// TIA Portal V18 export
// export: Created 2026-01-09T11:32:04.0903936Z, ExportSetting WithDefaults, DisplayName Totally Integrated Automation Portal, DisplayVersion V18 Update 5, DisplayName TIA Portal Openness, DisplayVersion V18 Update 5, DisplayName TIA Portal Teamcenter Gateway, DisplayVersion V18, DisplayName TIA Portal Version Control Interface, DisplayVersion V18, DisplayName SINAMICS Startdrive Advanced, DisplayVersion V18 SP2 Update 1, DisplayName SINAMICS Startdrive G110M, G120, G120C, G120D, G120P, G115D, DisplayVersion V18 SP2 Update 1, DisplayName SINAMICS Startdrive G130, G150, S120, S150, SINAMICS MV, S210, G220, S200, DisplayVersion V18 SP2 Update 1, DisplayName STEP 7 Professional, DisplayVersion V18 Update 5, DisplayName STEP 7 Safety, DisplayVersion V18, DisplayName WinCC Professional, DisplayVersion V18 Update 5
TagTable "ST_PM"
  ST_PMDBNum : Int  (1 s)
  ST_PMStepNext{1} : Bool  (%DB[ST_PMDBNum].DBX0.5, CPU S71500-2PN_TP700, 1 s)
  ST_PMStepNext{2} : Bool  (%DB[ST_PMDBNum].DBX20.5, CPU S71500-2PN_TP700, 1 s)
  ST_PMStepNext{3} : Bool  (%DB[ST_PMDBNum].DBX40.5, CPU S71500-2PN_TP700, 1 s)
  ST_PMStepNext{4} : Bool  (%DB[ST_PMDBNum].DBX60.5, CPU S71500-2PN_TP700, 1 s)
  ST_PMStepNext{5} : Bool  (%DB[ST_PMDBNum].DBX80.5, CPU S71500-2PN_TP700, 1 s)
  ST_PMStepNext{6} : Bool  (%DB[ST_PMDBNum].DBX100.5, CPU S71500-2PN_TP700, 1 s)
  ST_PMStepNext{7} : Bool  (%DB[ST_PMDBNum].DBX120.5, CPU S71500-2PN_TP700, 1 s)
  ST_PMStepNext{8} : Bool  (%DB[ST_PMDBNum].DBX140.5, CPU S71500-2PN_TP700, 1 s)
  ST_PMStepNext{9} : Bool  (%DB[ST_PMDBNum].DBX160.5, CPU S71500-2PN_TP700, 1 s)
  ST_PMStepNext{10} : Bool  (%DB[ST_PMDBNum].DBX180.5, CPU S71500-2PN_TP700, 1 s)
  ST_PMStepNext{11} : Bool  (%DB[ST_PMDBNum].DBX200.5, CPU S71500-2PN_TP700, 1 s)
  ST_PMStepNext{12} : Bool  (%DB[ST_PMDBNum].DBX220.5, CPU S71500-2PN_TP700, 1 s)
  ST_PMStepNext{13} : Bool  (%DB[ST_PMDBNum].DBX240.5, CPU S71500-2PN_TP700, 1 s)
  ST_PMStepNext{14} : Bool  (%DB[ST_PMDBNum].DBX260.5, CPU S71500-2PN_TP700, 1 s)
  ST_PMStepNext{15} : Bool  (%DB[ST_PMDBNum].DBX280.5, CPU S71500-2PN_TP700, 1 s)
  ST_PMStepNext{16} : Bool  (%DB[ST_PMDBNum].DBX300.5, CPU S71500-2PN_TP700, 1 s)
  ST_PMOperatorPrompt[0] : UInt  (%DB[ST_PMDBNum].DBW10, CPU S71500-2PN_TP700, 500 ms)
  ST_PMOperatorPrompt[1] : UInt  (%DB[ST_PMDBNum].DBW10, CPU S71500-2PN_TP700, 500 ms)
  ST_PMOperatorPrompt[2] : UInt  (%DB[ST_PMDBNum].DBW30, CPU S71500-2PN_TP700, 500 ms)
  ST_PMOperatorPrompt[3] : UInt  (%DB[ST_PMDBNum].DBW50, CPU S71500-2PN_TP700, 500 ms)
  ST_PMOperatorPrompt[4] : UInt  (%DB[ST_PMDBNum].DBW70, CPU S71500-2PN_TP700, 500 ms)
  ST_PMOperatorPrompt[5] : UInt  (%DB[ST_PMDBNum].DBW90, CPU S71500-2PN_TP700, 500 ms)
  ST_PMOperatorPrompt[6] : UInt  (%DB[ST_PMDBNum].DBW110, CPU S71500-2PN_TP700, 500 ms)
  ST_PMOperatorPrompt[7] : UInt  (%DB[ST_PMDBNum].DBW130, CPU S71500-2PN_TP700, 500 ms)
  ST_PMOperatorPrompt[8] : UInt  (%DB[ST_PMDBNum].DBW150, CPU S71500-2PN_TP700, 500 ms)
  ST_PMOperatorPrompt[9] : UInt  (%DB[ST_PMDBNum].DBW170, CPU S71500-2PN_TP700, 500 ms)
  ST_PMOperatorPrompt[10] : UInt  (%DB[ST_PMDBNum].DBW190, CPU S71500-2PN_TP700, 500 ms)
  ST_PMStep[11] : Int  (%DB[ST_PMDBNum].DBW214, CPU S71500-2PN_TP700, 100 ms)   // DBW00
  ST_PMStep[3] : Int  (%DB[ST_PMDBNum].DBW54, CPU S71500-2PN_TP700, 100 ms)   // DBW00
  ST_PMStep[14] : Int  (%DB[ST_PMDBNum].DBW274, CPU S71500-2PN_TP700, 100 ms)   // DBW00
  ST_PMStep[10] : Int  (%DB[ST_PMDBNum].DBW194, CPU S71500-2PN_TP700, 100 ms)   // DBW00
  ST_PMStep[8] : Int  (%DB[ST_PMDBNum].DBW154, CPU S71500-2PN_TP700, 100 ms)   // DBW00
  ST_PMStep[15] : Int  (%DB[ST_PMDBNum].DBW294, CPU S71500-2PN_TP700, 100 ms)   // DBW00
  ST_PMStep[13] : Int  (%DB[ST_PMDBNum].DBW254, CPU S71500-2PN_TP700, 100 ms)   // DBW00
  ST_PMStep[1] : Int  (%DB[ST_PMDBNum].DBW14, CPU S71500-2PN_TP700, 100 ms)   // DBW00
  ST_PMStep[12] : Int  (%DB[ST_PMDBNum].DBW234, CPU S71500-2PN_TP700, 100 ms)   // DBW00
  ST_PMStep[16] : Int  (%DB[ST_PMDBNum].DBW314, CPU S71500-2PN_TP700, 100 ms)   // DBW00
  ST_PMStep[2] : Int  (%DB[ST_PMDBNum].DBW34, CPU S71500-2PN_TP700, 100 ms)   // DBW00
  ST_PMStep[6] : Int  (%DB[ST_PMDBNum].DBW114, CPU S71500-2PN_TP700, 100 ms)   // DBW00
  ST_PMStep[4] : Int  (%DB[ST_PMDBNum].DBW74, CPU S71500-2PN_TP700, 100 ms)   // DBW00
  ST_PMStep[5] : Int  (%DB[ST_PMDBNum].DBW94, CPU S71500-2PN_TP700, 100 ms)   // DBW00
  ST_PMStep[7] : Int  (%DB[ST_PMDBNum].DBW134, CPU S71500-2PN_TP700, 100 ms)   // DBW00
  ST_PMStep[9] : Int  (%DB[ST_PMDBNum].DBW174, CPU S71500-2PN_TP700, 100 ms)   // DBW00
  ST_PMStep[30] : Int  (%DB[ST_PMDBNum].DBW594, CPU S71500-2PN_TP700, 1 s)
  ST_PMStep[29] : Int  (%DB[ST_PMDBNum].DBW574, CPU S71500-2PN_TP700, 1 s)
  ST_PMStep[28] : Int  (%DB[ST_PMDBNum].DBW554, CPU S71500-2PN_TP700, 1 s)
  ST_PMStep[27] : Int  (%DB[ST_PMDBNum].DBW534, CPU S71500-2PN_TP700, 1 s)
  ST_PMStep[26] : Int  (%DB[ST_PMDBNum].DBW514, CPU S71500-2PN_TP700, 1 s)
  ST_PMStep[25] : Int  (%DB[ST_PMDBNum].DBW494, CPU S71500-2PN_TP700, 1 s)
  ST_PMStep[24] : Int  (%DB[ST_PMDBNum].DBW474, CPU S71500-2PN_TP700, 1 s)
  ST_PMStep[23] : Int  (%DB[ST_PMDBNum].DBW454, CPU S71500-2PN_TP700, 1 s)
  ST_PMStep[22] : Int  (%DB[ST_PMDBNum].DBW434, CPU S71500-2PN_TP700, 1 s)
  ST_PMStep[21] : Int  (%DB[ST_PMDBNum].DBW414, CPU S71500-2PN_TP700, 1 s)
  ST_PMStep[20] : Int  (%DB[ST_PMDBNum].DBW394, CPU S71500-2PN_TP700, 1 s)
  ST_PMStep[19] : Int  (%DB[ST_PMDBNum].DBW374, CPU S71500-2PN_TP700, 1 s)
  ST_PMStep[18] : Int  (%DB[ST_PMDBNum].DBW354, CPU S71500-2PN_TP700, 1 s)
  ST_PMStep[17] : Int  (%DB[ST_PMDBNum].DBW334, CPU S71500-2PN_TP700, 1 s)
  ST_PMStepNext{17} : Bool  (%DB[ST_PMDBNum].DBX320.5, CPU S71500-2PN_TP700, 1 s)
  ST_PMStepNext{18} : Bool  (%DB[ST_PMDBNum].DBX340.5, CPU S71500-2PN_TP700, 1 s)
  ST_PMStepNext{19} : Bool  (%DB[ST_PMDBNum].DBX360.5, CPU S71500-2PN_TP700, 1 s)
  ST_PMStepNext{20} : Bool  (%DB[ST_PMDBNum].DBX380.5, CPU S71500-2PN_TP700, 1 s)
  ST_PMStepNext{21} : Bool  (%DB[ST_PMDBNum].DBX400.5, CPU S71500-2PN_TP700, 1 s)
  ST_PMStepNext{22} : Bool  (%DB[ST_PMDBNum].DBX420.5, CPU S71500-2PN_TP700, 1 s)
  ST_PMStepNext{23} : Bool  (%DB[ST_PMDBNum].DBX440.5, CPU S71500-2PN_TP700, 1 s)
  ST_PMStepNext{24} : Bool  (%DB[ST_PMDBNum].DBX460.5, CPU S71500-2PN_TP700, 1 s)
  ST_PMStepNext{25} : Bool  (%DB[ST_PMDBNum].DBX480.5, CPU S71500-2PN_TP700, 1 s)
  ST_PMStepNext{26} : Bool  (%DB[ST_PMDBNum].DBX500.5, CPU S71500-2PN_TP700, 1 s)
  ST_PMStepNext{27} : Bool  (%DB[ST_PMDBNum].DBX520.5, CPU S71500-2PN_TP700, 1 s)
  ST_PMStepNext{28} : Bool  (%DB[ST_PMDBNum].DBX540.5, CPU S71500-2PN_TP700, 1 s)
  ST_PMStepNext{29} : Bool  (%DB[ST_PMDBNum].DBX560.5, CPU S71500-2PN_TP700, 1 s)
  ST_PMStepNext{30} : Bool  (%DB[ST_PMDBNum].DBX580.5, CPU S71500-2PN_TP700, 1 s)
